# EPICS autosave request: optics/opticsApp/Db/2slit_settings.req
$(P)$(SLIT)xn_tweakVal
$(P)$(SLIT)xp_tweakVal
$(P)$(SLIT)size_tweakVal
$(P)$(SLIT)center_tweakVal
